(* CoDeSys 2.3.9.62 project: Mezcladora.pro *)
(* Libraries: Standard.lib 2.6.14 11:37:46, IecSfc.lib 2.6.14 10:37:46 *)

(* Task configuration *)
TASK NewTask (PRIORITY := 1, INTERVAL := T#100ms);
	PLC_PRG
END_TASK

(* Global variable list: Global_Variables *)
VAR_GLOBAL
   (* Entradas*)
    LInf: BOOL;
    LSup:BOOL;
    PS1:BOOL;
    PS2:BOOL;
    M:BOOL;
    P:BOOL;
    Emergencia:BOOL;
    Rearme:BOOL;

	Funciona:BOOL;
   (*Salidas*)
    LuzEm:BOOL;
   Valvula1:BOOL;
   Valvula2:BOOL;
   ValvulaA:BOOL;
   ValvulaB:BOOL;
   ValvulaC:BOOL;
   Motor:BOOL;

END_VAR

(* POU PLC_PRG, ST *)
PROGRAM PLC_PRG
VAR
END_VAR
MarchaParada;
Automatismo;
Depositos;
END_PROGRAM

(* POU MarchaParada, SFC *)
PROGRAM MarchaParada
VAR
END_VAR
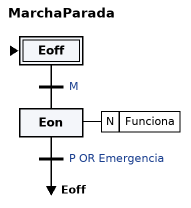
INITIAL_STEP Eoff:
END_STEP
TRANSITION FROM Eoff TO Eon := M;
END_TRANSITION
STEP Eon:
	Funciona(N);
END_STEP
TRANSITION FROM Eon TO Eoff := P OR Emergencia;
END_TRANSITION
END_PROGRAM

(* POU Automatismo, SFC *)
PROGRAM Automatismo
VAR
	Conta: CTU;
	RP:R_TRIG;
	ValP:BOOL;

END_VAR
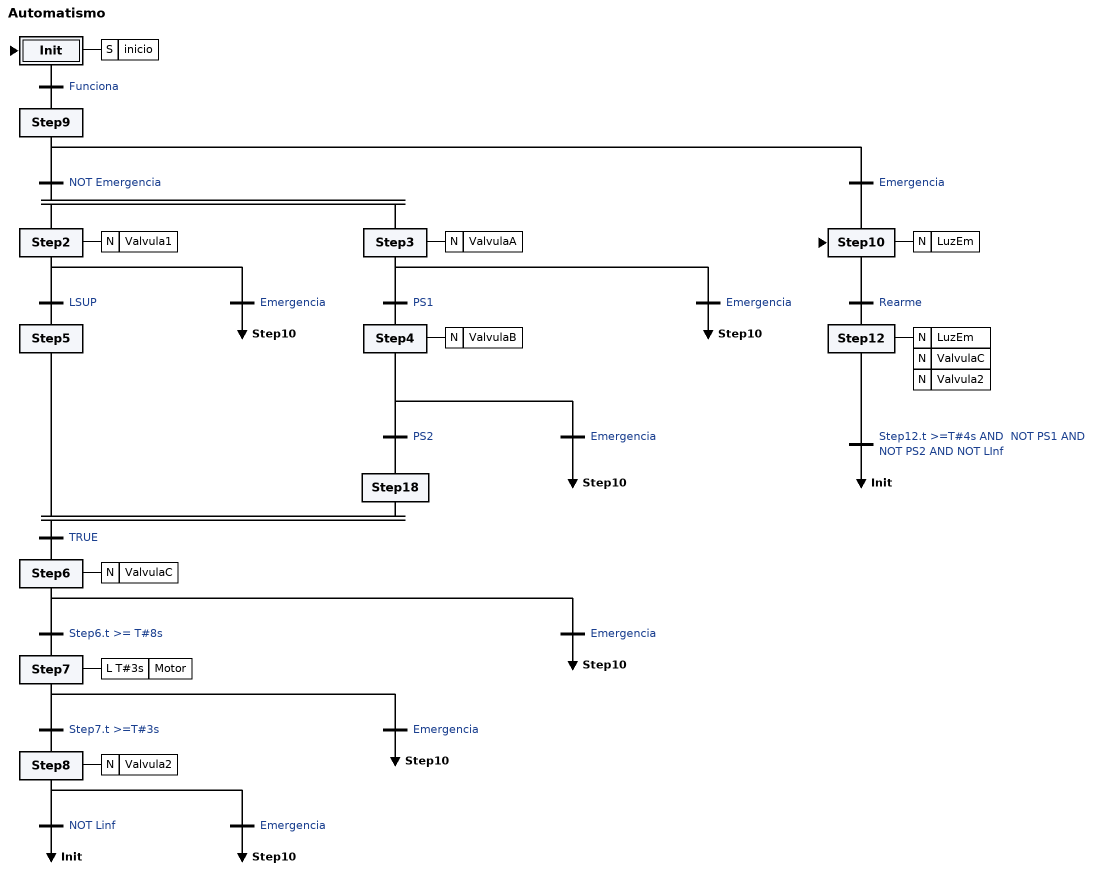
INITIAL_STEP Init:
	inicio(S);
END_STEP
TRANSITION FROM Init TO Step9 := Funciona;
END_TRANSITION
STEP Step9:
END_STEP
TRANSITION FROM Step9 TO (Step2, Step3) := NOT Emergencia;
END_TRANSITION
TRANSITION FROM Step9 TO Step10 := Emergencia;
END_TRANSITION
STEP Step10:
	LuzEm(N);
END_STEP
TRANSITION FROM Step10 TO Step12 := Rearme;
END_TRANSITION
STEP Step12:
	LuzEm(N);
	ValvulaC(N);
	Valvula2(N);
END_STEP
TRANSITION FROM Step12 TO Init := Step12.t >=T#4s AND  NOT PS1 AND NOT PS2 AND NOT LInf;
END_TRANSITION
STEP Step2:
	Valvula1(N);
END_STEP
TRANSITION FROM Step2 TO Step5 := LSUP;
END_TRANSITION
TRANSITION FROM Step2 TO Step10 := Emergencia;
END_TRANSITION
STEP Step5:
END_STEP
STEP Step3:
	ValvulaA(N);
END_STEP
TRANSITION FROM Step3 TO Step4 := PS1;
END_TRANSITION
TRANSITION FROM Step3 TO Step10 := Emergencia;
END_TRANSITION
STEP Step4:
	ValvulaB(N);
END_STEP
TRANSITION FROM Step4 TO Step18 := PS2;
END_TRANSITION
TRANSITION FROM Step4 TO Step10 := Emergencia;
END_TRANSITION
STEP Step18:
END_STEP
TRANSITION FROM (Step5, Step18) TO Step6 := TRUE;
END_TRANSITION
STEP Step6:
	ValvulaC(N);
END_STEP
TRANSITION FROM Step6 TO Step7 := Step6.t >= T#8s;
END_TRANSITION
TRANSITION FROM Step6 TO Step10 := Emergencia;
END_TRANSITION
STEP Step7:
	Motor(L, T#3s);
END_STEP
TRANSITION FROM Step7 TO Step8 := Step7.t >=T#3s;
END_TRANSITION
TRANSITION FROM Step7 TO Step10 := Emergencia;
END_TRANSITION
STEP Step8:
	Valvula2(N);
END_STEP
TRANSITION FROM Step8 TO Init := NOT Linf;
END_TRANSITION
TRANSITION FROM Step8 TO Step10 := Emergencia;
END_TRANSITION
END_PROGRAM
ACTION Inicio:
Conta(RESET:=P, CU:=Step8.x, PV:=3);(* el pv no sirve*)
END_ACTION

(* POU Depositos, ST *)
PROGRAM Depositos
VAR
   Nivel: REAL:=0.2;
   ValvulaEntrada:BOOL;
   ValvulaSalida:BOOL;
   CaudalEntrada:REAL:=0;
   CaudalSalida:REAL:=0;
   Area:REAL:=1;
   IntT:REAL:=0.1;
   KEntrada:REAL:=0.3;
   KSalida:REAL:=0.4;
	Neto: REAL;
	Nivellnf:REAL:=0;
	NivelSup:REAL:=2.2;
	CaudalEntrada2: REAL;
	CaudalSalida2: REAL;
	Neto2: REAL;
	Nivel2: REAL;
	Nivellnf2: REAL:=0;
	NivelSup2: REAL:=4;
	KSalida2: REAL:=0.8;
       Texto:STRING;
END_VAR
(*Deposito 1 *)
CaudalEntrada:=BOOL_TO_INT(Valvula1)*KEntrada;
CaudalSalida:=BOOL_TO_INT(Valvula2)*KSalida;
Neto:=(CaudalEntrada-CaudalSalida);
IF (Neto<0AND Nivel>Nivellnf) OR (Neto>0 AND Nivel<NivelSup) THEN
   Nivel:=Nivel+IntT*Neto;
END_IF

IF Nivel>0.33 THEN
   LInf:=TRUE;
ELSE
   LInf:=FALSE;
END_IF

IF Nivel>1.85 THEN
   LSup:=TRUE;
ELSE
   LSup:=FALSE;
END_IF

(*Deposito 2 *)
CaudalEntrada2:=(BOOL_TO_INT(ValvulaA)+BOOL_TO_INT(ValvulaB))*KEntrada;
CaudalSalida2:=BOOL_TO_INT(ValvulaC)*KSalida2;
Neto2:=(CaudalEntrada2-CaudalSalida2);
IF (Neto2<0AND Nivel2>Nivellnf2) OR (Neto2>0 AND Nivel2<NivelSup2) THEN
   Nivel2:=Nivel2+IntT*Neto2;
END_IF


IF Nivel2>2 THEN
   PS1:=TRUE;
ELSE
   PS1:=FALSE;
END_IF

IF Nivel2>3 THEN
   PS2:=TRUE;
ELSE
   PS2:=FALSE;
END_IF
END_PROGRAM

(* Visualisation Deposito
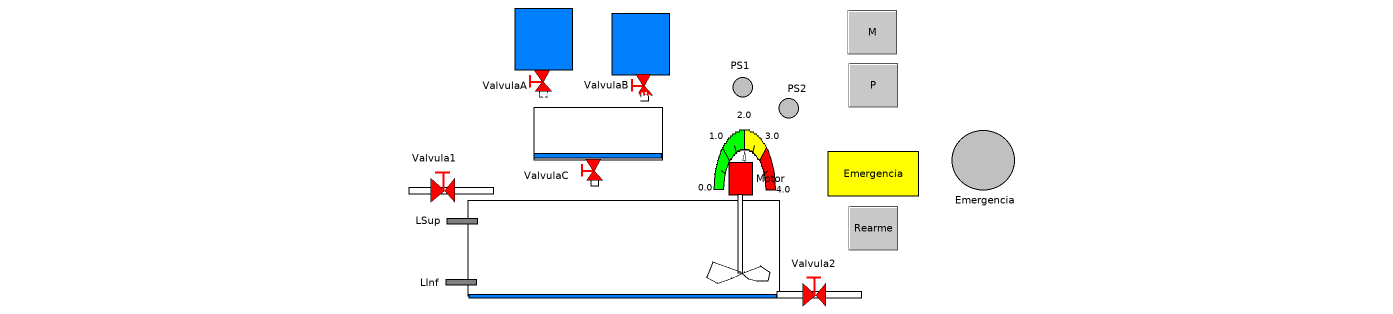
rectangle at (81,314)-(389,318): top -40*Depositos.Nivel
rectangle at (389,311)-(474,318): alarm colour if Valvula2 AND Depositos.Nivel>0
rectangle at (21,207)-(106,214): alarm colour if Valvula1
group at (43,192)-(67,222)
  polygon at (0,6)-(13,29): alarm colour if Valvula1
  polygon at (13,6)-(23,29): alarm colour if Valvula1
  polyline at (12,0)-(12,17): alarm colour if Valvula1
  polyline at (4,0)-(18,0): alarm colour if Valvula1
polygon at (415,303)-(428,326): alarm colour if Valvula2
polygon at (428,303)-(438,326): alarm colour if Valvula2
polyline at (427,297)-(427,314): alarm colour if Valvula2
polyline at (419,297)-(433,297): alarm colour if Valvula2
rectangle at (59,238)-(90,244): alarm colour if LSup
rectangle at (58,299)-(89,305): alarm colour if LInf
group at (142,90)-(164,117)
  polygon at (4,0)-(19,11): alarm colour if ValvulaA
  polygon at (5,11)-(21,21): alarm colour if ValvulaA
  polyline at (0,12)-(11,12): alarm colour if ValvulaA
  polyline at (0,5)-(0,17): alarm colour if ValvulaA
polygon at (248,94)-(263,105): alarm colour if ValvulaB
polygon at (249,105)-(265,115): alarm colour if ValvulaB
polyline at (244,106)-(255,106): alarm colour if ValvulaB
polyline at (244,99)-(244,111): alarm colour if ValvulaB
polygon at (198,179)-(213,190): alarm colour if ValvulaC
polygon at (199,190)-(215,200): alarm colour if ValvulaC
polyline at (194,191)-(205,191): alarm colour if ValvulaC
polyline at (194,184)-(194,196): alarm colour if ValvulaC
rectangle at (146,173)-(274,178): top -10*Depositos.Nivel2
group at (308,116)-(405,223)
  rectangle at (0,0)-(1,1): text "{ExtendedElement},Visu\ElementDLL.ete,0,@Zeigerinstrument,97,180,0,0,255,255,255,0,Depositos.Nivel2,,%.1f,0,1,1,0.5,1,0,4,0,0,0,0,0,0,0,-11,80,400,Arial,1,3,0,2,0,255,0,2,3,255,255,0,3,4,255,0,0,0,255,255,255,,0,0,0,0,"
  rectangle at (0,41)-(19,55): text "0.0"
  rectangle at (11,14)-(30,28): text "1.0"
  rectangle at (39,3)-(58,17): text "2.0"
  rectangle at (67,14)-(86,28): text "3.0"
  rectangle at (78,42)-(97,56): text "4.0"
  polygon at (47,29)-(50,49): angle ((Depositos.Nivel2 * 1.0)-2) * 45
ellipse at (345,97)-(365,117): alarm colour if PS1
ellipse at (391,118)-(411,138): alarm colour if PS2
rectangle at (20,160)-(72,196): text "Valvula1"
rectangle at (400,270)-(451,297): text "Valvula2"
rectangle at (90,90)-(144,121): text "ValvulaA"
rectangle at (190,89)-(247,121): text "ValvulaB"
rectangle at (130,180)-(187,211): text "ValvulaC"
rectangle at (334,70)-(371,101): text "PS1"
rectangle at (391,93)-(428,124): text "PS2"
rectangle at (23,287)-(60,318): text "LInf"
rectangle at (22,225)-(59,256): text "LSup"
rectangle at (341,182)-(365,215): alarm colour if Motor
rectangle at (364,183)-(401,214): text "Motor"
button at (460,30)-(509,74): text "M"; taps M
button at (461,83)-(510,127): text "P"; taps P
rectangle at (440,171)-(531,216): text "Emergencia"; alarm colour if Emergencia; taps Emergencia
button at (461,226)-(510,270): text "Rearme"; taps Rearme
ellipse at (564,150)-(627,210): alarm colour if LuzEm
rectangle at (550,200)-(644,240): text "Emergencia"
24 more shapes without text or variables
*)
